SUBAPPLICATION Uebung_225 (* Dreieck-Sollwertmarker: Sollwert-Eingabe bewegt das Dreieck und schreibt den Istwert zurueck *)
  (* Standard: 61499-2; Description: Copyright (c) 2026 Meisterschulen am Ostbahnhof This program and the accompanying materials are made available under the terms of the Eclipse Public License 2.0 which is available at https://www.eclipse.org/legal/epl-2.0/ SPDX-License-Identifier: EPL-2.0 *)
  (* Version 1.1, 2026-09-06, Franz Höpfinger, Meisterschulen am Ostbahnhof, Enable xScale on Q_ChildPosition_Dreieck *)
  (* Version 1.0, 2026-09-05, Franz Höpfinger, Meisterschulen am Ostbahnhof, initial API and implementation and/or initial documentation *)
  PACKAGE Uebungen;
  IMPORT Uebungen::const::UT::Dreieck::DefaultPool_Dreieck::Polygon_Bargraph_Mittelmarker;
  IMPORT Uebungen::const::UT::Dreieck::DefaultPool_Dreieck::Container_Sollwertmarker;
  IMPORT Uebungen::const::UT::Dreieck::DefaultPool_Dreieck_Numeric::NumberVariable_Sollwert_N;
  IMPORT Uebungen::const::UT::Dreieck::DefaultPool_Dreieck_Numeric::NumberVariable_Istwert_N;
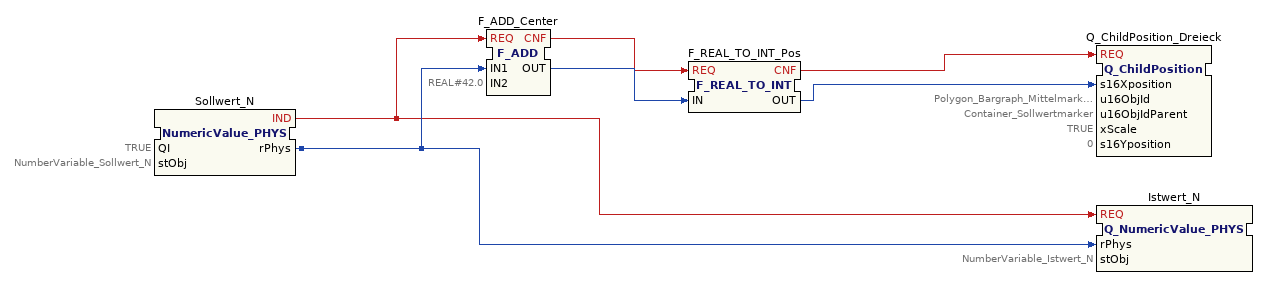
  FBS
    Sollwert_N : isobus::UT::io::NumericValue::NumericValue_PHYS(QI := TRUE, stObj := NumberVariable_Sollwert_N);
    F_ADD_Center : iec61131::arithmetic::F_ADD(IN2 := REAL#42.0);
    F_REAL_TO_INT_Pos : iec61131::conversion::F_REAL_TO_INT;
    Q_ChildPosition_Dreieck : isobus::UT::Q::Q_ChildPosition(u16ObjId := Polygon_Bargraph_Mittelmarker, u16ObjIdParent := Container_Sollwertmarker, xScale := TRUE, s16Yposition := 0);
    Istwert_N : isobus::UT::Q::Q_NumericValue_PHYS(stObj := NumberVariable_Istwert_N);
  END_FBS
  EVENT_CONNECTIONS
    Sollwert_N.IND TO F_ADD_Center.REQ;
    F_ADD_Center.CNF TO F_REAL_TO_INT_Pos.REQ;
    F_REAL_TO_INT_Pos.CNF TO Q_ChildPosition_Dreieck.REQ;
    Sollwert_N.IND TO Istwert_N.REQ;
  END_CONNECTIONS
  DATA_CONNECTIONS
    Sollwert_N.rPhys TO F_ADD_Center.IN1;
    F_ADD_Center.OUT TO F_REAL_TO_INT_Pos.IN;
    F_REAL_TO_INT_Pos.OUT TO Q_ChildPosition_Dreieck.s16Xposition;
    Sollwert_N.rPhys TO Istwert_N.rPhys;
  END_CONNECTIONS
END_SUBAPPLICATION
